SUBAPPLICATION Ventilsteuerung_Uebung_033 (* LED Strip Blinkende LED *)
  (* Standard: 61499-2 *)
  (* Version 1.0, 2023-10-23, franz *)
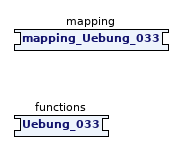
  SUBAPPS
    mapping : mapping_Uebung_033;
    functions : Uebung_033;
  END_SUBAPPS
END_SUBAPPLICATION
